# EPICS StreamDevice protocol: streamDevice/leds.proto
# Sidekick EPICS LEDs protocol file
# Built by examining examples at: https://paulscherrerinstitute.github.io/StreamDevice/protocol.html#gen

Terminator = CR LF;

info {
	ExtraInput = Ignore;
	out "*IDN?";
	in "%39c";
}

data {
	ExtraInput = Ignore;
	in "STREAM %39c";
}

# Brightness is an integer, 0 to 255
# Use long integer record type
getBrightness {
        out "BRIGhtness:LED\$1?";
        in "%u";
    }

setBrightness {
        out "BRIGhtness:LED\$1 %u";
        @init { getBrightness; }
    }

# Duration is an unsigned long integer
# Use int64 record type
getDuration {
        out "DURation:LED\$1?";
        in "%u";
    }

setDuration {
        out "DURation:LED\$1 %u";
        @init { getDuration; }
    }

# red
getRed {
		out "RED:LED\$1?";
		in "%f";
	}

setRed {
		out "RED:LED\$1 %f";
		@init { getRed; }
	}

# green
getGreen {
		out "GREEN:LED\$1?";
		in "%f";
	}

setGreen {
		out "GREEN:LED\$1 %f";
		@init { getGreen; }
	}

# blue
getBlue {
		out "BLUE:LED\$1?";
		in "%f";
	}

setBlue {
		out "BLUE:LED\$1 %f";
		@init { getBlue; }
	}

debug {
   ExtraInput = Ignore;
   out "%s";
   in "%39c";
}
